TYPE ST_TestBasicControl_out :
STRUCT
	DI0	: BOOL;
	out1	: DINT;
	out2	: DINT;
	stSub1Out	: ST_TestBasicControl_sub1;
	outStr1	: STRING(255);
	arrTest	: ARRAY[0..1] OF BYTE;
END_STRUCT
END_TYPE

(* stored: Version 1.1.0.1, ProductVersion 3.1.4024.9
   DUT ST_TestBasicControl_out: Id {1acaec01-869e-44de-9912-e090325ebd7d} *)
